Yaskawa INFORM job: X2_49(88,90).JBI

/JOB
//NAME X2_49(88,90)
//POS
///NPOS 187,187,187,11,0,0
///TOOL 0
///POSTYPE PULSE
///PULSE
C00000=2082,-130750,-111396,-32,62200,31
C00001=-101236,-103120,-120216,51408,79727,51679
C00002=-97957,-136705,-131009,52349,71210,48465
C00003=-97674,-104365,-117289,50526,76284,51543
C00004=-96811,-105247,-115474,50513,74807,51161
C00005=-96811,-105639,-114662,50651,74352,50906
C00006=-99566,-107368,-116035,51568,75801,50298
C00007=-99566,-107703,-115247,51689,75383,50056
C00008=-98124,-106686,-114889,51167,74797,50475
C00009=-99812,-107290,-116624,51575,76191,50392
C00010=-94397,-147158,-128591,53497,64933,46590
C00011=-92879,-140838,-124982,52724,64694,47345
C00012=-93366,-136489,-123755,52336,65893,47819
C00013=-94851,-142679,-125491,53469,65435,46644
C00014=-90811,-144101,-129314,51776,64145,48219
C00015=-94512,-129621,-125577,51241,69486,49344
C00016=-97957,-136705,-131009,52349,71210,48465
C00017=-97002,-130324,-129869,53153,76832,49930
C00018=-93420,-125545,-125031,52261,74511,50491
C00019=-93815,-118300,-120838,52151,75449,50830
C00020=-93815,-118530,-119843,52291,74989,50559
C00021=-97600,-121662,-121700,53409,76815,49589
C00022=-96939,-121270,-120539,53328,76129,49532
C00023=-95296,-119890,-120098,52810,75476,50040
C00024=-96939,-121270,-120539,53328,76129,49532
C00025=-97830,-129508,-124506,53882,75541,48676
C00026=-101579,-134301,-129310,54668,77990,48096
C00027=-96775,-130083,-130031,53052,76844,50061
C00028=-93202,-125317,-125195,52153,74528,50619
C00029=-93926,-117237,-120844,52082,75856,51010
C00030=-93926,-117493,-119930,52211,75420,50754
C00031=-98252,-120971,-122167,53473,77576,49697
C00032=-97501,-118998,-120261,53301,77058,49794
C00033=-95821,-117614,-119812,52771,76386,50306
C00034=-97501,-118998,-120261,53301,77058,49794
C00035=-98936,-116349,-121768,53346,79263,50350
C00036=-101813,-134411,-129545,54706,78178,48082
C00037=-96844,-129736,-130157,53028,77040,50142
C00038=-93273,-125036,-125337,52127,74713,50690
C00039=-94410,-117817,-121277,52230,76103,50896
C00040=-94410,-118032,-120527,52334,75744,50685
C00041=-98136,-120986,-122585,53406,77666,49817
C00042=-97004,-120312,-121169,53192,76708,49856
C00043=-95717,-119221,-120818,52783,76202,50253
C00044=-97004,-120312,-121169,53192,76708,49856
C00045=-97992,-129879,-125069,53889,75728,48702
C00046=-101750,-134681,-129872,54682,78179,48119
C00047=-90035,-147126,-129618,49072,53577,47593
C00048=-89817,-147839,-128607,49536,52799,47233
C00049=-90363,-147986,-127925,50043,52770,46867
C00050=-90363,-147443,-126977,50220,52571,46735
C00051=-94720,-152810,-129571,52506,54273,45066
C00052=-93566,-150613,-127666,52123,53590,45346
C00053=-91923,-148984,-127238,51190,53029,46034
C00054=-93566,-150613,-127666,52123,53590,45346
C00055=-96129,-155469,-133348,52464,55677,45124
C00056=-94726,-140540,-133485,47450,58991,49156
C00057=-120617,-140897,-132272,-714,58769,566
C00058=-146507,-141254,-131059,-48878,58548,-48024
C00059=-146507,-141254,-131059,-48878,58548,-48024
C00060=-149251,-130372,-124692,-46969,58248,-49410
C00061=-150278,-126561,-122251,-46309,58039,-49864
C00062=-150274,-126472,-120565,-46757,57346,-49480
C00063=-150278,-126561,-122251,-46309,58039,-49864
C00064=-144954,-132308,-122232,-49870,58832,-47288
C00065=-147637,-129972,-121538,-48443,57904,-48297
C00066=-144954,-132308,-122232,-49870,58832,-47288
C00067=-146870,-122472,-119531,-47621,60095,-49118
C00068=-145984,-116295,-117541,-47225,61899,-49629
C00069=-146870,-122472,-119531,-47621,60095,-49118
C00070=-145803,-125865,-121877,-48193,60449,-48726
C00071=-142965,-135301,-127915,-49791,61205,-47565
C00072=-144478,-130758,-130473,-52937,76607,-50110
C00073=-148050,-125868,-125604,-52026,74320,-50687
C00074=-149429,-123931,-123648,-51668,73428,-50908
C00075=-149425,-124118,-122047,-51910,72744,-50505
C00076=-149429,-123931,-123648,-51668,73428,-50908
C00077=-144777,-128798,-123401,-53494,74380,-48917
C00078=-147411,-126409,-122673,-52647,73371,-49772
C00079=-144777,-128798,-123401,-53494,74380,-48917
C00080=-143319,-130782,-125350,-53813,75321,-48680
C00081=-139556,-135784,-130204,-54614,77733,-48066
C00082=-144547,-131101,-130345,-52962,76411,-50030
C00083=-148121,-126146,-125460,-52053,74135,-50616
C00084=-149501,-124188,-123499,-51695,73246,-50841
C00085=-149497,-124346,-121889,-51938,72568,-50441
C00086=-149501,-124188,-123499,-51695,73246,-50841
C00087=-144709,-128567,-123082,-53526,74371,-48874
C00088=-147341,-126203,-122361,-52685,73356,-49724
C00089=-144709,-128567,-123082,-53526,74371,-48874
C00090=-143252,-130539,-125030,-53843,75315,-48639
C00091=-139492,-135504,-129875,-54638,77734,-48031
C00092=-144319,-131337,-130181,-53064,76400,-49899
C00093=-147902,-126370,-125294,-52162,74119,-50488
C00094=-149285,-124407,-123333,-51807,73228,-50714
C00095=-149282,-124537,-121714,-52049,72558,-50316
C00096=-149285,-124407,-123333,-51807,73228,-50714
C00097=-144934,-128413,-122833,-53488,74197,-48893
C00098=-147561,-126045,-122109,-52644,73186,-49744
C00099=-144934,-128413,-122833,-53488,74197,-48893
C00100=-143480,-130392,-124782,-53805,75138,-48657
C00101=-139727,-135378,-129635,-54600,77549,-48047
C00102=-143352,-137817,-131363,-52289,70764,-48425
C00103=-146796,-130512,-125878,-51157,69092,-49337
C00104=-143775,-111848,-117462,-51027,73584,-50305
C00105=-143775,-112183,-116375,-51211,73042,-49995
C00106=-143775,-112145,-116511,-51188,73108,-50034
C00107=-145087,-111128,-116162,-50693,72599,-50437
C00108=-143950,-131418,-123052,-52621,69285,-47859
C00109=-150539,-143690,-126535,-52180,62947,-47736
C00110=-150216,-141299,-124837,-52199,63246,-47733
C00111=-149440,-136363,-123449,-51798,64745,-48217
C00112=-148065,-145867,-126500,-53296,63653,-46701
C00113=-150539,-143690,-126535,-52180,62947,-47736
C00114=-145936,-129853,-123862,-51678,68993,-48799
C00115=-161026,-138216,-126703,-49813,63753,-51132
C00116=-161665,-136753,-124597,-49806,63049,-51079
C00117=-161065,-134227,-123929,-49673,63958,-51273
C00118=-161027,-138091,-126221,-49894,63601,-51043
C00119=-161027,-138117,-126319,-49877,63632,-51061
C00120=-160919,-138034,-125413,-50104,63353,-50834
C00121=-160827,-138180,-125479,-50145,63379,-50800
C00122=-161026,-138123,-126345,-49873,63640,-51066
C00123=-161026,-138149,-126443,-49855,63672,-51084
C00124=-160979,-137877,-125180,-50107,63279,-50827
C00125=-161031,-137790,-125134,-50083,63260,-50845
C00126=-161026,-138155,-126469,-49851,63680,-51089
C00127=-161026,-138180,-126567,-49834,63712,-51107
C00128=-161030,-137789,-125137,-50083,63262,-50846
C00129=-161030,-137791,-125143,-50082,63265,-50847
C00130=-161025,-138187,-126593,-49829,63720,-51112
C00131=-161025,-138211,-126691,-49812,63752,-51130
C00132=-161030,-137885,-125464,-50027,63362,-50905
C00133=-161030,-137913,-125556,-50011,63390,-50922
C00134=-161025,-138217,-126717,-49807,63760,-51135
C00135=-161025,-138241,-126815,-49790,63792,-51153
C00136=-161002,-137935,-125506,-50035,63375,-50899
C00137=-161029,-137910,-125551,-50012,63390,-50922
C00138=-161025,-138248,-126841,-49785,63800,-51158
C00139=-161024,-138271,-126938,-49768,63832,-51176
C00140=-161029,-137966,-125751,-49977,63453,-50956
C00141=-161115,-137805,-125614,-49950,63404,-50977
C00142=-161024,-138278,-126964,-49763,63841,-51181
C00143=-161024,-138301,-127062,-49746,63873,-51200
C00144=-161408,-137358,-125517,-49791,63355,-51115
C00145=-161317,-136919,-125443,-49754,63524,-51160
C00146=-161022,-138425,-127595,-49651,64048,-51301
C00147=-161007,-138954,-131130,-48996,65325,-52018
C00148=-161007,-147236,-133802,-48996,23562,-52018
C00149=-80310,-150896,-133802,61101,32496,52279
C00150=-160802,-137772,-129944,59373,113283,36180
C00151=-160803,-137161,-126386,58599,112280,35368
C00152=-161128,-135218,-123973,58374,112214,35097
C00153=-160970,-134558,-123803,58480,112245,35227
C00154=-160804,-137049,-125907,58501,112152,35266
C00155=-160804,-137071,-126004,58520,112178,35287
C00156=-161034,-134664,-124062,58516,112340,35259
C00157=-161113,-134576,-123997,58509,112392,35243
C00158=-160803,-137077,-126030,58525,112185,35292
C00159=-160803,-137100,-126127,58545,112211,35313
C00160=-161726,-135957,-124635,58326,112595,34987
C00161=-161461,-134428,-124288,58583,112741,35284
C00162=-160803,-137105,-126153,58550,112218,35318
C00163=-160803,-137127,-126250,58569,112244,35339
C00164=-161531,-135723,-124797,58433,112592,35119
C00165=-161283,-134547,-124483,58623,112664,35346
C00166=-160803,-137133,-126276,58574,112251,35345
C00167=-160802,-137155,-126373,58594,112277,35366
C00168=-161619,-135641,-125012,58495,112740,35174
C00169=-161479,-134137,-124752,58762,112987,35468
C00170=-160802,-137160,-126399,58599,112284,35371
C00171=-160802,-137181,-126496,58619,112310,35392
C00172=-161938,-136526,-125478,58393,112846,35039
C00173=-161650,-135460,-125171,58570,112863,35253
C00174=-160802,-137187,-126522,58624,112317,35398
C00175=-160801,-137208,-126618,58644,112343,35419
C00176=-161549,-135836,-125426,58564,112783,35255
C00177=-161401,-134739,-124981,58695,112850,35411
C00178=-160801,-137213,-126644,58649,112350,35425
C00179=-160801,-137233,-126741,58669,112376,35446
C00180=-162239,-139627,-126651,57997,112552,34605
C00181=-161518,-135008,-125307,58716,112953,35416
C00182=-160800,-137343,-127270,58778,112521,35562
C00183=-160799,-137822,-130790,59580,113542,36397
C00184=-62646,-142071,-133802,59580,113542,36397
C00185=-62646,-142071,-133802,59580,113542,36397
C00186=2082,-130750,-111396,-32,62200,31
BC00000=147868,666204,1075175
BC00001=266699,708353,1075175
BC00002=266699,754488,1075175
BC00003=266699,754488,1075175
BC00004=266699,754488,1075175
BC00005=266699,754488,1075175
BC00006=266699,754488,1075175
BC00007=266699,754488,1075175
BC00008=266699,754488,1075175
BC00009=266699,754488,1075175
BC00010=266699,754488,1075175
BC00011=266699,754488,1075175
BC00012=266699,754488,1075175
BC00013=266699,754488,1075175
BC00014=266699,754488,1075175
BC00015=266699,754488,1075175
BC00016=266699,754488,1075175
BC00017=264529,816560,1075175
BC00018=264529,816560,1075175
BC00019=264529,816560,1075175
BC00020=264529,816560,1075175
BC00021=264529,816560,1075175
BC00022=264529,816560,1075175
BC00023=264529,816560,1075175
BC00024=264529,816560,1075175
BC00025=264529,816560,1075175
BC00026=264529,816560,1075175
BC00027=265037,890074,1075175
BC00028=265037,890074,1075175
BC00029=265037,890074,1075175
BC00030=265037,890074,1075175
BC00031=265037,890074,1075175
BC00032=265037,890074,1075175
BC00033=265037,890074,1075175
BC00034=265037,890074,1075175
BC00035=265037,890074,1075175
BC00036=265037,890074,1075175
BC00037=265233,962169,1075175
BC00038=265233,962169,1075175
BC00039=265233,962169,1075175
BC00040=265233,962169,1075175
BC00041=265233,962169,1075175
BC00042=265233,962169,1075175
BC00043=265233,962169,1075175
BC00044=265233,962169,1075175
BC00045=265233,962169,1075175
BC00046=265233,962169,1075175
BC00047=270217,991120,1075175
BC00048=270217,991120,1075175
BC00049=270217,991120,1075175
BC00050=270217,991120,1075175
BC00051=270217,991120,1075175
BC00052=270217,991120,1075175
BC00053=270217,991120,1075175
BC00054=270217,991120,1075175
BC00055=270217,991120,1075175
BC00056=237014,944578,1075175
BC00057=220698,905523,1075175
BC00058=204382,943128,1075175
BC00059=168075,992313,1075175
BC00060=168075,992313,1075175
BC00061=168075,992313,1075175
BC00062=168075,992313,1075175
BC00063=168075,992313,1075175
BC00064=168075,992313,1075175
BC00065=168075,992313,1075175
BC00066=168075,992313,1075175
BC00067=168075,992313,1075175
BC00068=168075,992313,1075175
BC00069=168075,992313,1075175
BC00070=168075,992313,1075175
BC00071=168075,992313,1075175
BC00072=172728,963374,1075175
BC00073=172728,963374,1075175
BC00074=172728,963374,1075175
BC00075=172728,963374,1075175
BC00076=172728,963374,1075175
BC00077=172728,963374,1075175
BC00078=172728,963374,1075175
BC00079=172728,963374,1075175
BC00080=172728,963374,1075175
BC00081=172728,963374,1075175
BC00082=172446,891280,1075175
BC00083=172446,891280,1075175
BC00084=172446,891280,1075175
BC00085=172446,891280,1075175
BC00086=172446,891280,1075175
BC00087=172446,891280,1075175
BC00088=172446,891280,1075175
BC00089=172446,891280,1075175
BC00090=172446,891280,1075175
BC00091=172446,891280,1075175
BC00092=172467,817764,1075175
BC00093=172467,817764,1075175
BC00094=172467,817764,1075175
BC00095=172467,817764,1075175
BC00096=172467,817764,1075175
BC00097=172467,817764,1075175
BC00098=172467,817764,1075175
BC00099=172467,817764,1075175
BC00100=172467,817764,1075175
BC00101=172467,817764,1075175
BC00102=169910,755690,1075175
BC00103=169910,755690,1075175
BC00104=169910,755690,1075175
BC00105=169910,755690,1075175
BC00106=169910,755690,1075175
BC00107=169910,755690,1075175
BC00108=169910,755690,1075175
BC00109=169910,755690,1075175
BC00110=169910,755690,1075175
BC00111=169910,755690,1075175
BC00112=169910,755690,1075175
BC00113=169910,755690,1075175
BC00114=169910,755690,1075175
BC00115=185648,771444,1075175
BC00116=183829,771731,1075175
BC00117=183851,779412,1075175
BC00118=185540,779397,1075175
BC00119=185634,807960,1075175
BC00120=183945,807975,1075175
BC00121=183971,815655,1075175
BC00122=185660,815640,1075175
BC00123=185754,844203,1075175
BC00124=184065,844218,1075175
BC00125=184091,851898,1075175
BC00126=185780,851883,1075175
BC00127=185874,880446,1075175
BC00128=184185,880461,1075175
BC00129=184211,888141,1075175
BC00130=185900,888126,1075175
BC00131=185994,916689,1075175
BC00132=184305,916704,1075175
BC00133=184331,924384,1075175
BC00134=186020,924370,1075175
BC00135=186114,952932,1075175
BC00136=184425,952947,1075175
BC00137=184451,960627,1075175
BC00138=186140,960613,1075175
BC00139=186234,989176,1075175
BC00140=184545,989190,1075175
BC00141=184571,996870,1075175
BC00142=186260,996856,1075175
BC00143=186354,1025419,1075175
BC00144=184665,1025433,1075175
BC00145=184691,1033114,1075175
BC00146=186510,1032826,1075175
BC00147=191056,1032106,1075175
BC00148=191056,934026,1075175
BC00149=210326,796907,1075229
BC00150=330197,769559,1075175
BC00151=334751,770251,1075175
BC00152=336573,770528,1075175
BC00153=336603,778208,1075175
BC00154=334913,778204,1075175
BC00155=335007,806766,1075175
BC00156=336697,806771,1075171
BC00157=336723,814451,1075175
BC00158=335033,814447,1075175
BC00159=335127,843010,1075175
BC00160=336817,843014,1075175
BC00161=336843,850694,1075175
BC00162=335153,850690,1075175
BC00163=335247,879253,1075175
BC00164=336937,879257,1075175
BC00165=336963,886937,1075175
BC00166=335273,886933,1075175
BC00167=335367,915496,1075175
BC00168=337057,915500,1075175
BC00169=337083,923180,1075175
BC00170=335393,923176,1075175
BC00171=335487,951739,1075175
BC00172=337177,951743,1075175
BC00173=337203,959423,1075175
BC00174=335513,959419,1075175
BC00175=335607,987982,1075175
BC00176=337101,987986,1075175
BC00177=337323,995667,1075175
BC00178=335633,995662,1075175
BC00179=335727,1024225,1075175
BC00180=336885,1024228,1075172
BC00181=337367,1030745,1075175
BC00182=335621,1031633,1075175
BC00183=331067,1030941,1075175
BC00184=168360,888261,1075175
BC00185=168360,759459,1075175
BC00186=147868,666204,1075175
EC00000=780419,556475
EC00001=780419,556475
EC00002=780419,556475
EC00003=780419,556475
EC00004=780419,556475
EC00005=780419,556475
EC00006=780419,556475
EC00007=780419,556475
EC00008=780419,556475
EC00009=780419,556475
EC00010=780419,556475
EC00011=780419,556475
EC00012=780419,556475
EC00013=780419,556475
EC00014=780419,556475
EC00015=780419,556475
EC00016=780419,556475
EC00017=780419,556475
EC00018=780419,556475
EC00019=780419,556475
EC00020=780419,556475
EC00021=780419,556475
EC00022=780419,556475
EC00023=780419,556475
EC00024=780419,556475
EC00025=780419,556475
EC00026=780419,556475
EC00027=780419,556475
EC00028=780419,556475
EC00029=780419,556475
EC00030=780419,556475
EC00031=780419,556475
EC00032=780419,556475
EC00033=780419,556475
EC00034=780419,556475
EC00035=780419,556475
EC00036=780419,556475
EC00037=780419,556475
EC00038=780419,556475
EC00039=780419,556475
EC00040=780419,556475
EC00041=780419,556475
EC00042=780419,556475
EC00043=780419,556475
EC00044=780419,556475
EC00045=780419,556475
EC00046=780419,556475
EC00047=780419,556475
EC00048=780419,556475
EC00049=780419,556475
EC00050=780419,556475
EC00051=780419,556475
EC00052=780419,556475
EC00053=780419,556475
EC00054=780419,556475
EC00055=780419,556475
EC00056=780419,556475
EC00057=780419,556475
EC00058=780419,556475
EC00059=780419,556475
EC00060=780419,556475
EC00061=780419,556475
EC00062=780419,556475
EC00063=780419,556475
EC00064=780419,556475
EC00065=780419,556475
EC00066=780419,556475
EC00067=780419,556475
EC00068=780419,556475
EC00069=780419,556475
EC00070=780419,556475
EC00071=780419,556475
EC00072=780419,556475
EC00073=780419,556475
EC00074=780419,556475
EC00075=780419,556475
EC00076=780419,556475
EC00077=780419,556475
EC00078=780419,556475
EC00079=780419,556475
EC00080=780419,556475
EC00081=780419,556475
EC00082=780419,556475
EC00083=780419,556475
EC00084=780419,556475
EC00085=780419,556475
EC00086=780419,556475
EC00087=780419,556475
EC00088=780419,556475
EC00089=780419,556475
EC00090=780419,556475
EC00091=780419,556475
EC00092=780419,556475
EC00093=780419,556475
EC00094=780419,556475
EC00095=780419,556475
EC00096=780419,556475
EC00097=780419,556475
EC00098=780419,556475
EC00099=780419,556475
EC00100=780419,556475
EC00101=780419,556475
EC00102=780419,556475
EC00103=780419,556475
EC00104=780419,556475
EC00105=780419,556475
EC00106=780419,556475
EC00107=780419,556475
EC00108=780419,556475
EC00109=780419,556475
EC00110=780419,556475
EC00111=780419,556475
EC00112=780419,556475
EC00113=780419,556475
EC00114=780419,556475
EC00115=780419,556475
EC00116=780419,556475
EC00117=780419,556475
EC00118=780419,556475
EC00119=780419,556475
EC00120=780419,556475
EC00121=780419,556475
EC00122=780419,556475
EC00123=780419,556475
EC00124=780419,556475
EC00125=780419,556475
EC00126=780419,556475
EC00127=780419,556475
EC00128=780419,556475
EC00129=780419,556475
EC00130=780419,556475
EC00131=780419,556475
EC00132=780419,556475
EC00133=780419,556475
EC00134=780419,556475
EC00135=780419,556475
EC00136=780419,556475
EC00137=780419,556475
EC00138=780419,556475
EC00139=780419,556475
EC00140=780419,556475
EC00141=780419,556475
EC00142=780419,556475
EC00143=780419,556475
EC00144=780419,556475
EC00145=780419,556475
EC00146=780419,556475
EC00147=780419,556475
EC00148=780419,556475
EC00149=780419,556475
EC00150=780419,556475
EC00151=780419,556475
EC00152=780419,556475
EC00153=780419,556475
EC00154=780419,556475
EC00155=780419,556475
EC00156=780417,556475
EC00157=780419,556475
EC00158=780419,556475
EC00159=780419,556475
EC00160=780419,556475
EC00161=780419,556475
EC00162=780419,556475
EC00163=780419,556475
EC00164=780419,556475
EC00165=780419,556475
EC00166=780419,556475
EC00167=780419,556475
EC00168=780419,556475
EC00169=780419,556475
EC00170=780419,556475
EC00171=780419,556475
EC00172=780419,556475
EC00173=780419,556475
EC00174=780419,556475
EC00175=780419,556475
EC00176=780419,556475
EC00177=780419,556475
EC00178=780419,556475
EC00179=780419,556475
EC00180=780418,556475
EC00181=780419,556475
EC00182=780419,556475
EC00183=780419,556475
EC00184=780419,556475
EC00185=780419,556475
EC00186=780419,556475
///POSTYPE BASE
///RECTAN
///RCONF 0,0,0,0,0,0,0,0,0,0,0,0,0,0,0,0,0,0,0,0,0,0,0,0
P00006=0.222,-3.123,-1.508,0.0000,0.0000,0.0000
P00021=-0.225,-6.128,-0.405,0.0000,0.0000,0.0000
P00022=0.222,-3.123,-1.508,0.0000,0.0000,0.0000
P00023=0.143,-0.036,0.682,0.0000,0.0000,0.0000
P00024=0.145,-0.552,1.326,0.0000,0.0000,0.0000
P00025=-2.003,0.006,0.728,0.0000,0.0000,0.0000
P00031=1.853,-0.001,-1.549,0.0000,0.0000,0.0000
P00032=1.957,0.503,-7.217,0.0000,0.0000,0.0000
///RCONF 0,0,0,0,1,0,0,0,0,0,0,0,0,0,0,0,0,0,0,0,0,0,0,0
P00033=-0.123,0.612,-5.012,0.0000,0.0000,0.0000
///RCONF 0,0,0,0,0,0,0,0,0,0,0,0,0,0,0,0,0,0,0,0,0,0,0,0
P00034=-0.304,0.773,-2.693,0.0000,0.0000,0.0000
P00035=2.817,0.591,-1.622,0.0000,0.0000,0.0000
//INST
///DATE 2024/10/11 09:16
///ATTR SC,RW
///GROUP1 RB1,BS1
///GROUP2 ST1
NOP
'X2_49(88,90)
MOVJ C00000 BC00000 VJ=100.00  +MOVJ EC00000 VJ=100.00
MOVJ C00001 BC00001 VJ=100.00  +MOVJ EC00001 VJ=100.00
'Path S4716
SFTOF3D
MOVJ C00002 BC00002 VJ=100.00  +MOVJ EC00002 VJ=100.00
MOVL C00003 BC00003 V=800.0  +MOVJ EC00003 VJ=100.00
SMOVL C00004 BC00004 V=166.7  +MOVJ EC00004
SREFP 3 C00005 BC00005  +REFP EC00005
CALL JOB:SEARCH-R1-S13D
SET P031 P006
SFTON3D P031
SMOVL C00006 BC00006 V=166.7  +MOVJ EC00006
SMOVL C00007 BC00007 V=166.7  +MOVJ EC00007
SREFP 3 C00008 BC00008  +REFP EC00008
CALL JOB:SEARCH-R1-S13D
SET P031 P006
SFTON3D P031
SMOVL C00009 BC00009 V=166.7  +MOVJ EC00009
SMOVL C00010 BC00010 V=250.0  +MOVJ EC00010
SMOVL C00011 BC00011 V=166.7  +MOVJ EC00011
SREFP 3 C00012 BC00012  +REFP EC00012
CALL JOB:SEARCH-R1-S13D
SET P031 P006
SFTON3D P031
SMOVL C00013 BC00013 V=166.7  +MOVJ EC00013
SMOVL C00014 BC00014 V=250.0  +MOVJ EC00014
MOVL C00015 BC00015 V=800.0  +MOVJ EC00015 VJ=100.00
MOVL C00016 BC00016 V=1000.0  +MOVJ EC00016 VJ=100.00
'EndPath S4716
'Path S4715
SFTOF3D
MOVJ C00017 BC00017 VJ=100.00  +MOVJ EC00017 VJ=100.00
MOVL C00018 BC00018 V=800.0  +MOVJ EC00018 VJ=100.00
SMOVL C00019 BC00019 V=166.7  +MOVJ EC00019
SREFP 3 C00020 BC00020  +REFP EC00020
CALL JOB:SEARCH-R1-S13D
SET P032 P006
SFTON3D P032
SMOVL C00021 BC00021 V=166.7  +MOVJ EC00021
SMOVL C00022 BC00022 V=166.7  +MOVJ EC00022
SREFP 3 C00023 BC00023  +REFP EC00023
CALL JOB:SEARCH-R1-S13D
SET P032 P006
SFTON3D P032
SMOVL C00024 BC00024 V=166.7  +MOVJ EC00024
MOVL C00025 BC00025 V=800.0  +MOVJ EC00025 VJ=100.00
MOVL C00026 BC00026 V=1000.0  +MOVJ EC00026 VJ=100.00
'EndPath S4715
'Path S4714
SFTOF3D
MOVJ C00027 BC00027 VJ=100.00  +MOVJ EC00027 VJ=100.00
MOVL C00028 BC00028 V=800.0  +MOVJ EC00028 VJ=100.00
SMOVL C00029 BC00029 V=166.7  +MOVJ EC00029
SREFP 3 C00030 BC00030  +REFP EC00030
CALL JOB:SEARCH-R1-S13D
SET P033 P006
SFTON3D P033
SMOVL C00031 BC00031 V=166.7  +MOVJ EC00031
SMOVL C00032 BC00032 V=166.7  +MOVJ EC00032
SREFP 3 C00033 BC00033  +REFP EC00033
CALL JOB:SEARCH-R1-S13D
SET P033 P006
SFTON3D P033
SMOVL C00034 BC00034 V=166.7  +MOVJ EC00034
MOVL C00035 BC00035 V=800.0  +MOVJ EC00035 VJ=100.00
MOVL C00036 BC00036 V=1000.0  +MOVJ EC00036 VJ=100.00
'EndPath S4714
'Path S4713
SFTOF3D
MOVJ C00037 BC00037 VJ=100.00  +MOVJ EC00037 VJ=100.00
MOVL C00038 BC00038 V=800.0  +MOVJ EC00038 VJ=100.00
SMOVL C00039 BC00039 V=166.7  +MOVJ EC00039
SREFP 3 C00040 BC00040  +REFP EC00040
CALL JOB:SEARCH-R1-S13D
SET P034 P006
SFTON3D P034
SMOVL C00041 BC00041 V=166.7  +MOVJ EC00041
SMOVL C00042 BC00042 V=166.7  +MOVJ EC00042
SREFP 3 C00043 BC00043  +REFP EC00043
CALL JOB:SEARCH-R1-S13D
SET P034 P006
SFTON3D P034
SMOVL C00044 BC00044 V=166.7  +MOVJ EC00044
MOVL C00045 BC00045 V=800.0  +MOVJ EC00045 VJ=100.00
MOVL C00046 BC00046 V=1000.0  +MOVJ EC00046 VJ=100.00
'EndPath S4713
'Path S4712
SFTOF3D
MOVJ C00047 BC00047 VJ=100.00  +MOVJ EC00047 VJ=100.00
MOVL C00048 BC00048 V=800.0  +MOVJ EC00048 VJ=100.00
SMOVL C00049 BC00049 V=166.7  +MOVJ EC00049
SREFP 3 C00050 BC00050  +REFP EC00050
CALL JOB:SEARCH-R1-S13D
SET P035 P006
SFTON3D P035
SMOVL C00051 BC00051 V=166.7  +MOVJ EC00051
SMOVL C00052 BC00052 V=166.7  +MOVJ EC00052
SREFP 3 C00053 BC00053  +REFP EC00053
CALL JOB:SEARCH-R1-S13D
SET P035 P006
SFTON3D P035
SMOVL C00054 BC00054 V=166.7  +MOVJ EC00054
MOVL C00055 BC00055 V=1000.0  +MOVJ EC00055 VJ=100.00
'EndPath S4712
MOVJ C00056 BC00056 VJ=100.00  +MOVJ EC00056 VJ=100.00
MOVJ C00057 BC00057 VJ=100.00  +MOVJ EC00057 VJ=100.00
MOVJ C00058 BC00058 VJ=100.00  +MOVJ EC00058 VJ=100.00
'Path S4295
SFTOF3D
MOVJ C00059 BC00059 VJ=100.00  +MOVJ EC00059 VJ=100.00
MOVL C00060 BC00060 V=800.0  +MOVJ EC00060 VJ=100.00
SMOVL C00061 BC00061 V=166.7  +MOVJ EC00061
SREFP 3 C00062 BC00062  +REFP EC00062
CALL JOB:SEARCH-R1-S13D
SET P025 P006
SFTON3D P025
SMOVL C00063 BC00063 V=166.7  +MOVJ EC00063
SMOVL C00064 BC00064 V=166.7  +MOVJ EC00064
SREFP 3 C00065 BC00065  +REFP EC00065
CALL JOB:SEARCH-R1-S13D
SET P025 P006
SFTON3D P025
SMOVL C00066 BC00066 V=166.7  +MOVJ EC00066
SMOVL C00067 BC00067 V=166.7  +MOVJ EC00067
SREFP 3 C00068 BC00068  +REFP EC00068
CALL JOB:SEARCH-R1-S13D
SET P025 P006
SFTON3D P025
SMOVL C00069 BC00069 V=166.7  +MOVJ EC00069
MOVL C00070 BC00070 V=800.0  +MOVJ EC00070 VJ=100.00
MOVL C00071 BC00071 V=1000.0  +MOVJ EC00071 VJ=100.00
'EndPath S4295
'Path S4296
SFTOF3D
MOVJ C00072 BC00072 VJ=100.00  +MOVJ EC00072 VJ=100.00
MOVL C00073 BC00073 V=800.0  +MOVJ EC00073 VJ=100.00
SMOVL C00074 BC00074 V=166.7  +MOVJ EC00074
SREFP 3 C00075 BC00075  +REFP EC00075
CALL JOB:SEARCH-R1-S13D
SET P024 P006
SFTON3D P024
SMOVL C00076 BC00076 V=166.7  +MOVJ EC00076
SMOVL C00077 BC00077 V=166.7  +MOVJ EC00077
SREFP 3 C00078 BC00078  +REFP EC00078
CALL JOB:SEARCH-R1-S13D
SET P024 P006
SFTON3D P024
SMOVL C00079 BC00079 V=166.7  +MOVJ EC00079
MOVL C00080 BC00080 V=800.0  +MOVJ EC00080 VJ=100.00
MOVL C00081 BC00081 V=1000.0  +MOVJ EC00081 VJ=100.00
'EndPath S4296
'Path S4297
SFTOF3D
MOVJ C00082 BC00082 VJ=100.00  +MOVJ EC00082 VJ=100.00
MOVL C00083 BC00083 V=800.0  +MOVJ EC00083 VJ=100.00
SMOVL C00084 BC00084 V=166.7  +MOVJ EC00084
SREFP 3 C00085 BC00085  +REFP EC00085
CALL JOB:SEARCH-R1-S13D
SET P023 P006
SFTON3D P023
SMOVL C00086 BC00086 V=166.7  +MOVJ EC00086
SMOVL C00087 BC00087 V=166.7  +MOVJ EC00087
SREFP 3 C00088 BC00088  +REFP EC00088
CALL JOB:SEARCH-R1-S13D
SET P023 P006
SFTON3D P023
SMOVL C00089 BC00089 V=166.7  +MOVJ EC00089
MOVL C00090 BC00090 V=800.0  +MOVJ EC00090 VJ=100.00
MOVL C00091 BC00091 V=1000.0  +MOVJ EC00091 VJ=100.00
'EndPath S4297
'Path S4298
SFTOF3D
MOVJ C00092 BC00092 VJ=100.00  +MOVJ EC00092 VJ=100.00
MOVL C00093 BC00093 V=800.0  +MOVJ EC00093 VJ=100.00
SMOVL C00094 BC00094 V=166.7  +MOVJ EC00094
SREFP 3 C00095 BC00095  +REFP EC00095
CALL JOB:SEARCH-R1-S13D
SET P022 P006
SFTON3D P022
SMOVL C00096 BC00096 V=166.7  +MOVJ EC00096
SMOVL C00097 BC00097 V=166.7  +MOVJ EC00097
SREFP 3 C00098 BC00098  +REFP EC00098
CALL JOB:SEARCH-R1-S13D
SET P022 P006
SFTON3D P022
SMOVL C00099 BC00099 V=166.7  +MOVJ EC00099
MOVL C00100 BC00100 V=800.0  +MOVJ EC00100 VJ=100.00
MOVL C00101 BC00101 V=1000.0  +MOVJ EC00101 VJ=100.00
'EndPath S4298
'Path S3705
SFTOF3D
MOVJ C00102 BC00102 VJ=100.00  +MOVJ EC00102 VJ=100.00
MOVL C00103 BC00103 V=800.0  +MOVJ EC00103 VJ=100.00
SMOVL C00104 BC00104 V=166.7  +MOVJ EC00104
SREFP 3 C00105 BC00105  +REFP EC00105
CALL JOB:SEARCH-R1-S13D
SET P021 P006
SFTON3D P021
SMOVL C00106 BC00106 V=166.7  +MOVJ EC00106
SREFP 3 C00107 BC00107  +REFP EC00107
CALL JOB:SEARCH-R1-S13D
SET P021 P006
SFTON3D P021
SMOVL C00108 BC00108 V=166.7  +MOVJ EC00108
SMOVL C00109 BC00109 V=166.7  +MOVJ EC00109
SMOVL C00110 BC00110 V=166.7  +MOVJ EC00110
SREFP 3 C00111 BC00111  +REFP EC00111
CALL JOB:SEARCH-R1-S13D
SET P021 P006
SFTON3D P021
SMOVL C00112 BC00112 V=166.7  +MOVJ EC00112
SMOVL C00113 BC00113 V=166.7  +MOVJ EC00113
SMOVL C00114 BC00114 V=166.7  +MOVJ EC00114
'EndPath S3705
'Path W3708
SFTOF3D
SFTON3D P021
SMOVL C00115 BC00115 V=800.0  +MOVJ EC00115
SMOVL C00116 BC00116 V=150.0 PL=0  +MOVJ EC00116
MACRO1 MJ#(0) ARGF9
ARCON
SMOVL C00117 BC00117 V=12.5  +MOVJ EC00117
ARCOF
SMOVL C00118 BC00118 V=150.0  +MOVJ EC00118
SFTON3D P022
SMOVL C00119 BC00119 V=150.0  +MOVJ EC00119
SMOVL C00120 BC00120 V=150.0 PL=0  +MOVJ EC00120
ARCON
SMOVL C00121 BC00121 V=12.5  +MOVJ EC00121
ARCOF
SMOVL C00122 BC00122 V=150.0  +MOVJ EC00122
SMOVL C00123 BC00123 V=150.0  +MOVJ EC00123
SMOVL C00124 BC00124 V=150.0 PL=0  +MOVJ EC00124
ARCON
SMOVL C00125 BC00125 V=12.5  +MOVJ EC00125
ARCOF
SMOVL C00126 BC00126 V=150.0  +MOVJ EC00126
SFTON3D P023
SMOVL C00127 BC00127 V=150.0  +MOVJ EC00127
SMOVL C00128 BC00128 V=150.0 PL=0  +MOVJ EC00128
ARCON
SMOVL C00129 BC00129 V=12.5  +MOVJ EC00129
ARCOF
SMOVL C00130 BC00130 V=150.0  +MOVJ EC00130
SMOVL C00131 BC00131 V=150.0  +MOVJ EC00131
SMOVL C00132 BC00132 V=150.0 PL=0  +MOVJ EC00132
ARCON
SMOVL C00133 BC00133 V=12.5  +MOVJ EC00133
ARCOF
SMOVL C00134 BC00134 V=150.0  +MOVJ EC00134
SFTON3D P024
SMOVL C00135 BC00135 V=150.0  +MOVJ EC00135
SMOVL C00136 BC00136 V=150.0 PL=0  +MOVJ EC00136
ARCON
SMOVL C00137 BC00137 V=12.5  +MOVJ EC00137
ARCOF
SMOVL C00138 BC00138 V=150.0  +MOVJ EC00138
SMOVL C00139 BC00139 V=150.0  +MOVJ EC00139
SMOVL C00140 BC00140 V=150.0 PL=0  +MOVJ EC00140
ARCON
SMOVL C00141 BC00141 V=12.5  +MOVJ EC00141
ARCOF
SMOVL C00142 BC00142 V=150.0  +MOVJ EC00142
SFTON3D P025
SMOVL C00143 BC00143 V=150.0  +MOVJ EC00143
SMOVL C00144 BC00144 V=150.0 PL=0  +MOVJ EC00144
ARCON
SMOVL C00145 BC00145 V=12.5  +MOVJ EC00145
ARCOF
SMOVL C00146 BC00146 V=800.0  +MOVJ EC00146
SMOVL C00147 BC00147 V=1000.0  +MOVJ EC00147
SFTOF3D
'EndPath W3708
MOVJ C00148 BC00148 VJ=100.00  +MOVJ EC00148 VJ=100.00
MOVJ C00149 BC00149 VJ=100.00  +MOVJ EC00149 VJ=100.00
'Path W4711
SFTOF3D
SFTON3D P031
MOVJ C00150 BC00150 VJ=100.00  +MOVJ EC00150 VJ=100.00
SMOVL C00151 BC00151 V=800.0  +MOVJ EC00151
SMOVL C00152 BC00152 V=150.0 PL=0  +MOVJ EC00152
ARCON
SMOVL C00153 BC00153 V=12.5  +MOVJ EC00153
ARCOF
SMOVL C00154 BC00154 V=150.0  +MOVJ EC00154
SFTON3D P032
SMOVL C00155 BC00155 V=150.0  +MOVJ EC00155
SMOVL C00156 BC00156 V=150.0 PL=0  +MOVJ EC00156
ARCON
SMOVL C00157 BC00157 V=12.5  +MOVJ EC00157
ARCOF
SMOVL C00158 BC00158 V=150.0  +MOVJ EC00158
SMOVL C00159 BC00159 V=150.0  +MOVJ EC00159
SMOVL C00160 BC00160 V=150.0 PL=0  +MOVJ EC00160
ARCON
SMOVL C00161 BC00161 V=12.5  +MOVJ EC00161
ARCOF
SMOVL C00162 BC00162 V=150.0  +MOVJ EC00162
SFTON3D P033
SMOVL C00163 BC00163 V=150.0  +MOVJ EC00163
SMOVL C00164 BC00164 V=150.0 PL=0  +MOVJ EC00164
ARCON
SMOVL C00165 BC00165 V=12.5  +MOVJ EC00165
ARCOF
SMOVL C00166 BC00166 V=150.0  +MOVJ EC00166
SMOVL C00167 BC00167 V=150.0  +MOVJ EC00167
SMOVL C00168 BC00168 V=150.0 PL=0  +MOVJ EC00168
ARCON
SMOVL C00169 BC00169 V=12.5  +MOVJ EC00169
ARCOF
SMOVL C00170 BC00170 V=150.0  +MOVJ EC00170
SFTON3D P034
SMOVL C00171 BC00171 V=150.0  +MOVJ EC00171
SMOVL C00172 BC00172 V=150.0 PL=0  +MOVJ EC00172
ARCON
SMOVL C00173 BC00173 V=12.5  +MOVJ EC00173
ARCOF
SMOVL C00174 BC00174 V=150.0  +MOVJ EC00174
SMOVL C00175 BC00175 V=150.0  +MOVJ EC00175
SMOVL C00176 BC00176 V=150.0 PL=0  +MOVJ EC00176
ARCON
SMOVL C00177 BC00177 V=12.5  +MOVJ EC00177
ARCOF
SMOVL C00178 BC00178 V=150.0  +MOVJ EC00178
SFTON3D P035
SMOVL C00179 BC00179 V=150.0  +MOVJ EC00179
SMOVL C00180 BC00180 V=150.0 PL=0  +MOVJ EC00180
ARCON
SMOVL C00181 BC00181 V=12.5  +MOVJ EC00181
ARCOF
SMOVL C00182 BC00182 V=800.0  +MOVJ EC00182
SMOVL C00183 BC00183 V=1000.0  +MOVJ EC00183
SFTOF3D
'EndPath W4711
MOVJ C00184 BC00184 VJ=100.00  +MOVJ EC00184 VJ=100.00
MOVJ C00185 BC00185 VJ=100.00  +MOVJ EC00185 VJ=100.00
MOVJ C00186 BC00186 VJ=100.00  +MOVJ EC00186 VJ=100.00
END
